PROGRAM MAIN
VAR
	
		fb_S_UPS	:	FB_S_UPS;
		
		fbEcatDiag1	:	FB_EcatDiag;
		fbEcatDiag2 :	FB_EcatDiag;
	
END_VAR



//fb_S_UPS.iPLCPort := AMSPORT_R0_PLC_RTS2;
fb_S_UPS(iPLCPort:=851);


p_modbusRx();

p_Autosave();

p_ESTOP();

fbEcatDiag1(i_AMSNetId:=g_aEcatMaster1, i_xFirstPass:=g_xFirstPass, q_xAllStatesGood=>g_xIOState);
fbEcatDiag2(i_AMSNetId:=g_aEcatMaster2, i_xFirstPass:=g_xFirstPass, q_xAllStatesGood=>g_xIOState);

p_SoftIO();

//p_SelectorDetector();

p_SampleSelector();
p_SampleSelector2();
p_Regulators();
p_Shakers();
p_Manifold();
p_ALI();
//p_VacGaugeSup();


//p_CoolerShaker();

p_ModbusTx();

p_StatusLights();

(* Following execution of all the programs, set the first pass false *)
g_xFirstPass := FALSE;

END_PROGRAM

(* stored: Version 1.1.0.1, ProductVersion 3.1.4018.5
   POU MAIN: Id {42c5d645-8f72-4a7d-9897-ab636f1cee6d}, SpecialFunc None *)
